FUNCTION_BLOCK FB_System_Ampel
VAR_INPUT
	Freigabe_auto			: BOOL;
	Betrieb_Anford_auto		: BOOL;
	Regelung_Sollw_auto		: ST_System_Ampel_Signal;
END_VAR
VAR_OUTPUT
	{attribute 'OPC.UA.DA' := '1'}Steuerung				: ST_System_Ampel_Steuerung;		
	{attribute 'OPC.UA.DA' := '1'}Stellwert				: ST_System_Ampel_Stellwert;		
	{attribute 'OPC.UA.DA' := '1'}Zustand					: ST_System_Ampel_Zustand;		
END_VAR
VAR
	Signal_Ampel: FB_Ampel;
	Sollwertscheck: FB_System_Ampel_Sollwertscheck;
END_VAR

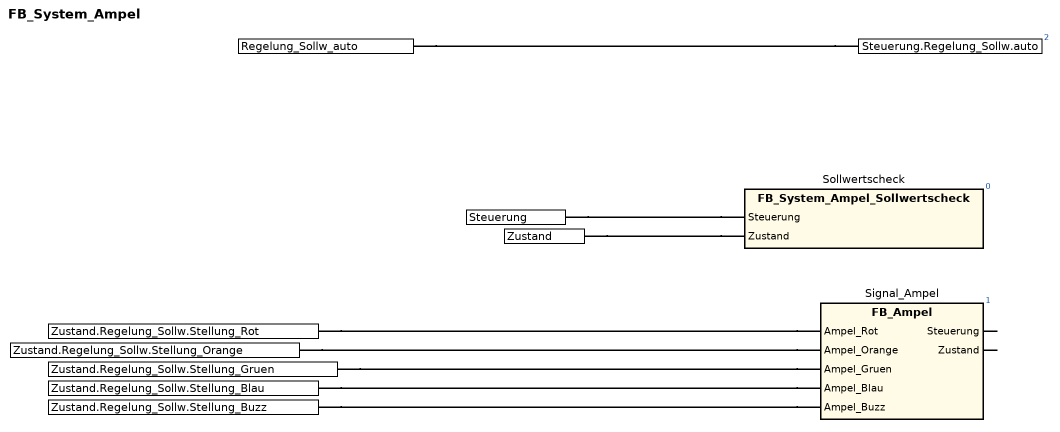
Sollwertscheck(Steuerung := Steuerung, Zustand := Zustand); // FB_System_Ampel_Sollwertscheck
Signal_Ampel(
    Ampel_Rot := Zustand.Regelung_Sollw.Stellung_Rot,
    Ampel_Orange := Zustand.Regelung_Sollw.Stellung_Orange,
    Ampel_Gruen := Zustand.Regelung_Sollw.Stellung_Gruen,
    Ampel_Blau := Zustand.Regelung_Sollw.Stellung_Blau,
    Ampel_Buzz := Zustand.Regelung_Sollw.Stellung_Buzz); // FB_Ampel
Steuerung.Regelung_Sollw.auto := Regelung_Sollw_auto;

END_FUNCTION_BLOCK

(* stored: Version 1.1.0.1, ProductVersion 3.1.4024.9
   POU FB_System_Ampel: Id {57d7b339-fddb-434c-8b0b-ea7376269bfd}, SpecialFunc None *)
